PROGRAM MQTTComm
VAR
END_VAR

END_PROGRAM

(* stored: Version 1.1.0.1, ProductVersion 3.1.4022.9
   POU MQTTComm: Id {efe7e652-d626-4d55-97a9-285f5546527a}, SpecialFunc None *)
